SYSTEM TESTBED_VIEWL (* Testbed View + HMI *)
  (* Standard: 61499 ITA; Classification: Testbed *)
  (* Version 0.3, 2004-10-26, JHC, Rockwell Automation, Changed rotary representation to gate on ring chute. *)
  (* Version 0.2, 2004-10-22, JHC, Rockwell Automation, Reformatted XSPACEs to work with DIA=40 or 25.. *)
  (* Version 0.1, 2004-09-28, JHC, Rockwell Automation, Updated for new conveyor models. *)
  (* Version 0.0, 2002-04-15, JHC, Rockwell Automation *)
  DEVICE HMI : FRAME_DEVICE(BOUNDS := [100,100,375,360], GRID := [1,1])
    RESOURCE HMI_PANEL : PANEL_RESOURCE
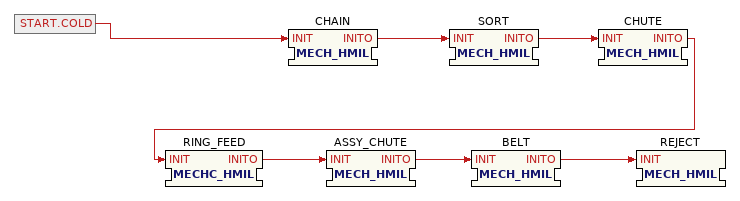
      FBS
        CHAIN : MECH_HMIL;
        SORT : MECH_HMIL;
        CHUTE : MECH_HMIL;
        RING_FEED : MECHC_HMIL;
        ASSY_CHUTE : MECH_HMIL;
        BELT : MECH_HMIL;
        REJECT : MECH_HMIL;
      END_FBS
      EVENT_CONNECTIONS
        START.COLD TO CHAIN.INIT;
        CHAIN.INITO TO SORT.INIT;
        CHUTE.INITO TO RING_FEED.INIT;
        RING_FEED.INITO TO ASSY_CHUTE.INIT;
        SORT.INITO TO CHUTE.INIT;
        BELT.INITO TO REJECT.INIT;
        ASSY_CHUTE.INITO TO BELT.INIT;
      END_CONNECTIONS
    END_RESOURCE
  END_DEVICE
  DEVICE MODEL : FRAME_DEVICE(BOUNDS := [475,100,290,360])
    RESOURCE CHAIN : VIEW_PANEL(DIA := 40, SIZE := [7,2])
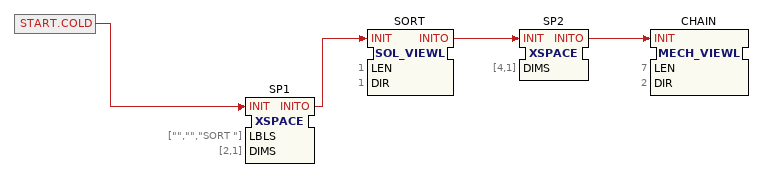
      FBS
        SP1 : XSPACE(LBLS := ["","","SORT "], DIMS := [2,1]);
        SORT : SOL_VIEWL(LEN := 1, DIR := 1); (* Sort Solenoid *)
        SP2 : XSPACE(DIMS := [4,1]);
        CHAIN : MECH_VIEWL(LEN := 7, DIR := 2); (* First Chain Segment *)
      END_FBS
      EVENT_CONNECTIONS
        START.COLD TO SP1.INIT;
        SP1.INITO TO SORT.INIT;
        SORT.INITO TO SP2.INIT;
        SP2.INITO TO CHAIN.INIT;
      END_CONNECTIONS
    END_RESOURCE
    RESOURCE CHUTES : VIEW_PANEL(DIA := 40, SIZE := [7,4], VERTICAL := 1)
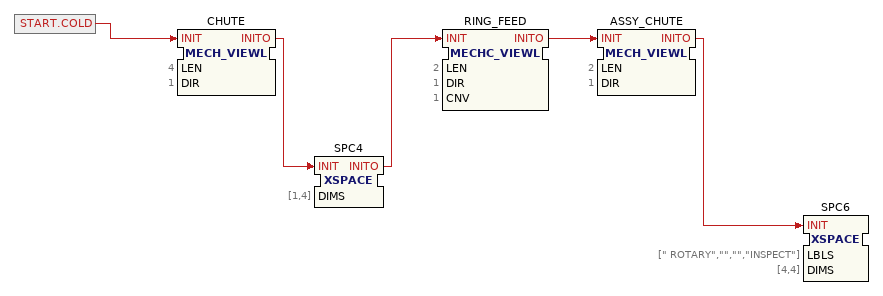
      FBS
        CHUTE : MECH_VIEWL(LEN := 4, DIR := 1); (* Peg Chute *)
        SPC4 : XSPACE(DIMS := [1,4]); (* Ring Feed Chute *)
        RING_FEED : MECHC_VIEWL(LEN := 2, DIR := 1, CNV := 1); (* Ring Feed Chute *)
        ASSY_CHUTE : MECH_VIEWL(LEN := 2, DIR := 1); (* Assembly Chute *)
        SPC6 : XSPACE(LBLS := [" ROTARY","","","INSPECT"], DIMS := [4,4]);
      END_FBS
      EVENT_CONNECTIONS
        START.COLD TO CHUTE.INIT;
        CHUTE.INITO TO SPC4.INIT;
        SPC4.INITO TO RING_FEED.INIT;
        RING_FEED.INITO TO ASSY_CHUTE.INIT;
        ASSY_CHUTE.INITO TO SPC6.INIT;
      END_CONNECTIONS
    END_RESOURCE
    RESOURCE BELT : VIEW_PANEL(DIA := 40, SIZE := [7,2])
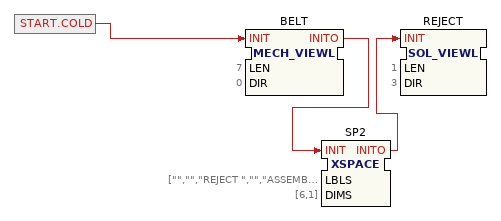
      FBS
        BELT : MECH_VIEWL(LEN := 7, DIR := 0);
        SP2 : XSPACE(LBLS := ["","","REJECT ","","ASSEMBLE"], DIMS := [6,1]);
        REJECT : SOL_VIEWL(LEN := 1, DIR := 3);
      END_FBS
      EVENT_CONNECTIONS
        START.COLD TO BELT.INIT;
        SP2.INITO TO REJECT.INIT;
        BELT.INITO TO SP2.INIT;
      END_CONNECTIONS
    END_RESOURCE
  END_DEVICE
END_SYSTEM
